(*udt (user defined type) of Beckhoff EL1908 - 8 Point PNP Safety Type Input Terminal:
	June 2014;*)


TYPE udt_EP1908_002 :
STRUCT
	I: BYTE;

	InfoData: udt_ECATSlave_Status;
END_STRUCT
END_TYPE

(* stored: Version 1.1.0.1, ProductVersion 3.1.4024.9
   DUT udt_EP1908_002: Id {56a6689c-5c34-49ee-aa63-113c909fd9c9} *)
